INTERFACE I_Telescope

PROPERTY AltAz : ST_AltAzCoordinate
GET
END_GET
END_PROPERTY

METHOD ABSTRACT Home : BOOL
VAR_INPUT
END_VAR
END_METHOD

METHOD MoveAltAz : BOOL
VAR_INPUT
	AltAz	: ST_AltAzCoordinate;
END_VAR
END_METHOD

METHOD MoveRaDec : BOOL
VAR_INPUT
	RaDec	: ST_RaDecCoordinate;
END_VAR
END_METHOD

METHOD ABSTRACT Park : BOOL
VAR_INPUT
END_VAR
END_METHOD

METHOD ABSTRACT PowerOff : BOOL
VAR_INPUT
END_VAR
END_METHOD

METHOD ABSTRACT PowerOn : BOOL
VAR_INPUT
END_VAR
END_METHOD

PROPERTY RaDec : ST_RaDecCoordinate
GET
END_GET
END_PROPERTY

METHOD Reset : BOOL
VAR_INPUT
END_VAR
END_METHOD

METHOD SetAltitudeOffset : BOOL
VAR_INPUT
	Offset	: LREAL;
END_VAR
END_METHOD

METHOD SetAzimuthOffset : BOOL
VAR_INPUT
	Offset	: LREAL;
END_VAR
END_METHOD

METHOD SetDerotatorOffset : BOOL
VAR_INPUT
	Offset	: LREAL;
END_VAR
END_METHOD

METHOD Stop : BOOL
VAR_INPUT
END_VAR
END_METHOD

METHOD TrackRaDec : BOOL
VAR_INPUT
	RaDec	: ST_RaDecCoordinate;
END_VAR
END_METHOD

END_INTERFACE

(* stored: Version 1.1.0.1, ProductVersion 3.1.4024.13
   Itf I_Telescope: Id {5003d6e3-4b52-4cb8-a028-b0ab2a6b3370}
   Property AltAz: Id {a6146940-4650-466d-9ac9-c2c5b727745a}
   Get Get: Id {8ad68625-dc7b-4361-8150-63f54617c376}
   Method Home: Id {2fc689c7-e332-49bc-87f2-069b41e58195}
   Method MoveAltAz: Id {cc0d567e-4a90-40d9-8f8e-e1a94eb43aa2}
   Method MoveRaDec: Id {3fa8011d-980e-4e74-a2b5-1fdb3dd84098}
   Method Park: Id {4989c55f-52d0-4389-8fa2-916073e653f8}
   Method PowerOff: Id {3291b764-646f-4fe2-b792-3aa38b38e854}
   Method PowerOn: Id {22b1f0f6-3e21-43e9-a91c-d9db89f97e54}
   Property RaDec: Id {12c8886c-56f7-4ec9-a493-221526805c02}
   Get Get: Id {d3f2ced6-23ed-44bd-a553-0d3cbd87919b}
   Method Reset: Id {7c6108fb-54b5-48bf-af67-cc7170330ed5}
   Method SetAltitudeOffset: Id {1a4df7a8-72ea-47ad-923c-f0c163cab97c}
   Method SetAzimuthOffset: Id {03e900b7-1d08-4452-a79c-3f3c7fce3a8a}
   Method SetDerotatorOffset: Id {4321acfd-c2aa-4930-a9a9-411c79360413}
   Method Stop: Id {078c3ad2-bc5e-4ad8-9b03-f137aaad29d9}
   Method TrackRaDec: Id {17caa4eb-aef5-4541-b247-843b6eb5de40} *)
